{attribute 'global_init_slot' := '40600'}
VAR_GLOBAL CONSTANT
	{attribute 'global_init_slot'}
	DiMouduleMAX 			:	INT	:=	10;
	{attribute 'global_init_slot'}
	DOMODULEMAX 			:	INT	:=	10;
	{attribute 'global_init_slot'}
	SiMouduleMAX 			:	INT	:=	10;
	{attribute 'global_init_slot'}
	SoMODULEMAX 			:	INT	:=	10;	
END_VAR

VAR_GLOBAL
	arDI	AT%I*		: ARRAY[0..DiMouduleMAX ] OF ST_IO_16;		//  links to Digital input  Modules 
	arDO	AT%Q*		: ARRAY[0..DOMODULEMAX ] OF ST_IO_16;		//  links to Digital output Modules	
	arSI	AT%I*		: ARRAY[0..SiMouduleMAX ] OF ST_SafetyIO;	//  links to safety input  Modules
	arSO	AT%I*		: ARRAY[0..SOMODULEMAX ] OF ST_SafetyIO;	//  links to safety output  Modules
END_VAR

(* stored: Version 1.1.0.1, ProductVersion 3.1.4024.12
   GVL G_IO: Id {dfe05562-cd77-4d74-a229-ed718eb42956} *)
